FUNCTION F_Azimuthvelocity : LREAL
VAR_INPUT
	// elevation in degrees
	elevation: 	LREAL;
	// azimuth in degrees
	azimuth:	LREAL;
	// observers latitude in degrees
	latitude:	LREAL;
END_VAR
VAR
END_VAR

IF ABS(COS(elevation * GVL_Math.d2r))> 1.0e-3 THEN
	F_Azimuthvelocity := (SIN(latitude * GVL_Math.d2r) - COS(latitude * GVL_Math.d2r) * COS(azimuth * GVL_Math.d2r) * TAN(elevation * GVL_Math.d2r))* GVL_Math.Omega;
ELSE
	F_Azimuthvelocity := 0.0;	
END_IF

END_FUNCTION

(* stored: Version 1.1.0.1, ProductVersion 3.1.4024.15
   POU F_Azimuthvelocity: Id {82607675-d3a6-495f-a7ca-8160127ea6de}, SpecialFunc None *)
